FUNCTION_BLOCK POU EXTENDS FB_ReadEL6688CoE
VAR_INPUT
END_VAR
VAR_OUTPUT
END_VAR
VAR
END_VAR

END_FUNCTION_BLOCK

(* stored: Version 1.1.0.1, ProductVersion 3.1.4022.12
   POU POU: Id {354f178c-7dbb-4aed-971f-daafe37d283e}, SpecialFunc None *)
